{attribute 'linkalways'} 
{attribute 'no_explicit_call' := 'This FB is a CLASS and must be accessed using methods or properties'}
{attribute 'enable_dynamic_creation'}
FUNCTION_BLOCK GearOutCommand EXTENDS Mc2Command
VAR
	fb : Tc2_Mc2.Mc_GearOut;
END_VAR

METHOD PUBLIC CyclicCall
SUPER^.CyclicCall();
fb(Slave := axis_ref);
END_METHOD

METHOD PROTECTED OnExecuting
VAR_INPUT
	state_control : AsyncCommandStateControl;
END_VAR
fb.Execute := TRUE;

IF fb.Done THEN
	state_control.Next();
	fb.Execute := FALSE;
END_IF

IF fb.Error THEN
	state_control.Error(fb.ErrorId);
	fb.Execute := FALSE;
END_IF
END_METHOD

END_FUNCTION_BLOCK

(* stored: Version 1.1.0.1
   POU GearOutCommand: Id {ccf50e5d-7079-0445-1476-280f83d53bc1}, SpecialFunc None
   Method CyclicCall: Id {cb026375-1154-0afb-3a48-e67b9645e989}
   Method OnExecuting: Id {97d197df-2bd1-09da-0357-323ac344c517} *)
